FUNCTION_BLOCK ADSReadBasic
VAR_INPUT
END_VAR
VAR_OUTPUT
END_VAR
VAR
	AdsRead : ADSREAD;
	rtrig : R_TRIG;
	ReadState : INT;
	_Busy : BOOL;
	_done : BOOL;
END_VAR

//Sequence
CASE ReadState OF
	0://Wait for Read Command
		IF rtrig.Q THEN
			_done := FALSE;
			_Busy := TRUE;
			AdsRead.READ := TRUE;
			ReadState := 10;
		END_IF
	10://Wait for read busy
		IF AdsRead.BUSY THEN
			ReadState := 20;
		END_IF
	20://Wait for execute finish
		IF NOT AdsRead.BUSY THEN
			_Busy := FALSE;
			_done := true;
			AdsRead.READ := FALSE;
			rtrig.CLK := FALSE;
			ReadState := 0;
		END_IF
END_CASE

//Outputs

//FBs
rtrig();
AdsRead(TMOUT := T#5S);

PROPERTY Busy : BOOL
GET
Busy := THIS^._Busy;
END_GET
END_PROPERTY

PROPERTY Done : BOOL
GET
Done := _done;
END_GET
END_PROPERTY

{warning 'add property implementation'}
PROPERTY Error : BOOL
GET
Error := AdsRead.ERR;
END_GET
END_PROPERTY

{warning 'add property implementation'}
PROPERTY ErrorId : UDINT
GET
ErrorId := AdsRead.ERRID;
END_GET
END_PROPERTY

METHOD PUBLIC Execute : BOOL
VAR_INPUT
END_VAR
 IF NOT rtrig.CLK THEN
	 rtrig.CLK := true;
 END_IF
END_METHOD

METHOD PUBLIC SetADSReadTarget : BOOL
VAR_INPUT
	TargetNetId     : T_AmsNetId;
    TargetPort      : T_AmsPort;
    AdsIdxGrp    : UDINT;
    AdsIdxOff   : UDINT;
    ReadLength       : UDINT;
    ReadVarAddr  : PVOID;	
END_VAR
AdsRead.DESTADDR := ReadVarAddr;
AdsRead.IDXGRP := AdsIdxGrp;
AdsRead.IDXOFFS := AdsIdxOff;
AdsRead.LEN := ReadLength;
AdsRead.NETID := TargetNetId;
AdsRead.PORT := TargetPort;
END_METHOD

END_FUNCTION_BLOCK

(* stored: Version 1.1.0.1, ProductVersion 3.1.4024.12
   POU ADSReadBasic: Id {0ffe9e63-1be4-478e-95e1-bcfdc1358ff7}, SpecialFunc None
   Property Busy: Id {682f512b-183c-4a93-9244-aa2a70d83e38}
   Get Get: Id {f9d5266e-78d3-4100-b386-c27b9870d325}
   Property Done: Id {dce508fd-599c-4458-8815-2339dd23e2c0}
   Get Get: Id {cd0f783a-b08e-4a79-85c3-3b87bd34d6dc}
   Property Error: Id {d8eed527-635f-498b-bd98-d5582534bf44}
   Get Get: Id {103f2642-8799-4c0b-b481-1f6932314715}
   Property ErrorId: Id {e5c429b5-4c36-4239-97b2-0585e498513c}
   Get Get: Id {89b589ed-8869-4a6c-8319-114d30b8b065}
   Method Execute: Id {8663fbcd-01ed-497d-a9cb-e4bbfca9b8dd}
   Method SetADSReadTarget: Id {457af66e-c705-4e7d-a3ed-92d52625251b} *)
